FUNCTION_BLOCK FB_ShapeCreatorEX EXTENDS FB_ShapeCreator
VAR_INPUT
END_VAR
VAR_OUTPUT
END_VAR
VAR
	pCustomShape : POINTER TO FB_CustomShape;
END_VAR

METHOD M_GetShapeObject : I_shape
VAR_INPUT
END_VAR
IF eShape = E_Shape.Custom THEN
	
	//Dynamic instantiation  
	pCustomShape := __NEW(FB_CustomShape);
	iShape := pCustomShape^;
	
	//Return the object
	IF iShape <> 0 THEN
		M_GetShapeObject := iShape;
	END_IF
	
	//Release the memory
	IF (pCustomShape <> 0) THEN
		__DELETE(pCustomShape);
		pCustomShape := 0;
	END_IF
	
	eShape := E_Shape.init;
ELSE
	M_GetShapeObject := SUPER^.M_GetShapeObject();
END_IF
END_METHOD

END_FUNCTION_BLOCK

(* stored: Version 1.1.0.1, ProductVersion 3.1.4024.12
   POU FB_ShapeCreatorEX: Id {93f27fe8-d1f0-42c5-bf70-f6fa273e98d5}, SpecialFunc None
   Method M_GetShapeObject: Id {c401e67d-4bf3-4a6d-87a8-2f37fb7f54ac} *)
